// TwinCAT 3 PLC project PLC
// ProgramVersion: 3.1.4026.12
// CompilerDefines: VISU_USEPROPERTYINFO
// libraries:
//   Tc2_MC2, * (Beckhoff Automation GmbH)
//   Tc2_SPA, * (Beckhoff Automation GmbH)
//   Tc2_Standard, * (Beckhoff Automation GmbH)
//   Tc2_System, * (Beckhoff Automation GmbH)
//   Tc2_Utilities, * (Beckhoff Automation GmbH)
//   VisuSymbols, 4.5.0.0 (System)
// project tree:
//   / GlobalTextList.TcGTLO, PlcTask.TcTTO, Visualization Manager.TcVMO (not stored)
//   GVLs/ GVL.TcGVL
//   POUs/ FB_PositionMotors.TcPOU, FB_PyListener.TcPOU, MAIN.TcPOU
//   VISUs/ Visualization.TcVIS
// real-time tasks:
//   TASK PlcTask: cycle T#10ms, priority 20, ADS port 350
// motion (NC):
//   TASK NC-Task 1 SAF: cycle T#2ms, priority 4, ADS port 501
//   TASK NC-Task 1 SVB: cycle T#10ms, priority 8, ADS port 511
//   AXIS Az (id 1)
//     General: UnitName=°, UnitFlags=#x00000004
//     OtherSettings: AllowMotionCmdToSlave=true
//     encoder EncType=1
//       Inc: RefSoftSyncMask=#x0000ffff
//     drive DrvType=5
//       Analog: TorqueSetpointScale=10, ScaleFactorActTorque=0.1
//       TimeComp: TaskDelayCycles=1
//     controller CtrType=1
//       CtrPara: PriorControlFactor=1
//         Observer: BandWidth=20
//   AXIS Alt (id 2)
//     General: UnitName=°, UnitFlags=#x00000004
//     PositionAreaControl: Enable=false
//     TargetPosControl: Enable=false
//     encoder EncType=1
//       SoftEndMinControl: Enable=true
//       SoftEndMaxControl: Enable=true, Range=90
//       Inc: RefSoftSyncMask=#x0000ffff
//     drive DrvType=5
//       Analog: TorqueSetpointScale=10, ScaleFactorActTorque=0.1
//       TimeComp: TaskDelayCycles=1
//     controller CtrType=1
//       CtrPara: PriorControlFactor=1
//         PosDiffControl: Enable=false
//         Observer: BandWidth=20
// I/O:
//   DEVICE Device 1 (EtherCAT), AmsNetId 192.168.1.5.2.1
//     Term 1 (EK1100) [EK1100 EtherCAT Coupler (2A E-Bus)]
//       Term 2 (EL7041) [EL7041 1Ch. Stepper motor output stage (50V, 5A)] (disabled)
//       Term 3 (EL7041) [EL7041 1Ch. Stepper motor output stage (50V, 5A)] (disabled)
// variable links:
//   PLC/PLC Instance <-> NC-Task 1 SAF/Axes/Alt
//     PlcTask Inputs/GVL.Alt.NcToPlc <-> Outputs/ToPlc
//     PlcTask Outputs/GVL.Alt.PlcToNc <-> Inputs/FromPlc
//   PLC/PLC Instance <-> NC-Task 1 SAF/Axes/Az
//     PlcTask Inputs/GVL.Az.NcToPlc <-> Outputs/ToPlc
//     PlcTask Outputs/GVL.Az.PlcToNc <-> Inputs/FromPlc

CONFIGURATION PLC
    RESOURCE PLC ON TwinCAT3
        TASK PlcTask(INTERVAL := T#10ms, PRIORITY := 20);
        PROGRAM MAIN WITH PlcTask : MAIN;
    END_RESOURCE
END_CONFIGURATION

// ---- GVLs/GVL.TcGVL
{attribute 'qualified_only'}
VAR_GLOBAL
	Alt				: Axis_Ref := Alt;
	Az				: Axis_Ref := Az;
END_VAR

// ---- POUs/MAIN.TcPOU
PROGRAM MAIN
VAR
	// Sun position variables
	fbGetTime				: NT_GetTime;
	fbPyListener			: FB_PyListener;
	currTime				: TIMESTRUCT;
	timer					: TON;
	fbSPA     				: FB_SPA;
    fSunZenith 				: LREAL;
    fSunAzimuth 			: LREAL;
	fSunAltitude			: LREAL;
    tSunrise    			: TIME;
    tSunset     			: TIME;
    eErrorCode 				: E_SPA_ErrorCode;
    bExecute    			: BOOL := TRUE;
    bInit     				: BOOL := TRUE;
	go						: BOOL := FALSE;
	
	// Motion control variables
	fbPositionMotors		: FB_PositionMotors;
	fbResetMotors			: MC_Reset;
	bResetMotors			: BOOL := FALSE;
	Az						: Axis_Ref;
	Alt						: Axis_Ref;
	
END_VAR

timer(
	IN := TRUE, 
	PT := T#1S
	);

fbGetTime(
	NETID := '',
	Start := timer.Q,
	TMOUT := DEFAULT_ADS_TIMEOUT,
	BUSY =>,
	ERRID =>,
	TIMESTR => currTime
	);
	
fbPylistener(bExecute := TRUE);					// Grab lat, long, and other data... tell the rest of the
												// program when its done and its good to go

IF timer.Q THEN
 	fbSPA.stTime.iYear := currTime.wYear;
 	fbSPA.stTime.iMonth := currTime.wMonth;
 	fbSPA.stTime.iDay := currtime.wDay;
 	fbSPA.stTime.iHour := currTime.wHour;
 	fbSPA.stTime.iMinute := currTime.wMinute;
 	fbSPA.fTimezone; 							// Uses UTC offset
 	fbSPA.fLongitude; 							// Grabbed from Python script
 	fbSPA.fLatitude; 							// Grabbed from Python script
 	fbSPA.fElevation; 							// Meters, grabbed from Python script
 	fbSPA.fTemperature := 20; 					// Celsius... grab temp from either web, python, USB, or whatever
 	fbSPA.eFunction := eSPA_ZA_RTS;
END_IF

IF go = TRUE THEN 								// Tie all GO commands to execute after geo location 
												// is found, Q timers

IF timer.Q THEN
	
    fbSPA();
	
    fSunZenith := fbSPA.fZenith;
	fSunAltitude := 90 - fSunZenith; 			// Get altitude from zenith
    fSunAzimuth := fbSPA.fAzimuth;
    tSunrise := LREAL_TO_TIME(fbSPA.fSunrise * 60 * 60 * 1000);
    tSunset := LREAL_TO_TIME(fbSPA.fSunset * 60 * 60 * 1000);
	
	eErrorCode := fbSPA.iErrorCode;
	
	fbPositionMotors( 
		fSunAltitude := fSunAltitude,
		fSunAzimuth := fSunAzimuth 
		);
	
	IF bResetMotors = TRUE THEN
		fbResetMotors(Axis := GVL.Az, Execute := TRUE);
		fbResetMotors(Axis := GVL.Alt, Execute := TRUE);
		bResetMotors := FALSE;
	END_IF
	
END_IF

IF (timer.Q) THEN
	timer(IN := FALSE);
END_IF

END_IF

END_PROGRAM

// ---- POUs/FB_PyListener.TcPOU
FUNCTION_BLOCK FB_PyListener
VAR_INPUT
	bExecute			: BOOL := FALSE;
	Initialized 		: BOOL := FALSE;
	Init_State  		: UINT := 0;
END_VAR
VAR_OUTPUT
	bIsBusy				: BOOL;
    ERR             	: BOOL;
    ERRID           	: UDINT;
END_VAR
VAR
	Process         	: NT_StartProcess;
	RisingEdge			: R_TRIG;
	bError          	: BOOL;
    sTargetFilePath     : STRING(255);
    sTargetDirectory    : STRING(255);
    sCommand        	: STRING(255);
    iErrorId            : UDINT; 	
END_VAR

IF NOT Initialized THEN
  (* Initialization State Machine *)
  CASE Init_State OF
    0: (* First step in initialization *)
	
		// File Locations
		sTargetDirectory := 'C:\Users\AEverman\Desktop\Celestial_Positioning\Celestial_Positioning\Celestial_Positioning\PLC\SCRIPTS\';
 
		// Build Command String                 
		// Special command indicating command string input
		sCommand := CONCAT(sTargetDirectory, 'GPS_COORD_FIND.py');      // Execute Python data collection script
        Init_State := Init_State + 1;
	   
    1: (* Second step in initialization *)
		Process(
    	NETID := '',                    					// Local System
		//PATHSTR := 'C:\ProgramData\Anaconda3\python.exe ',   // Path to local cmd executable
		PATHSTR := 'python',
    	COMNDLINE := sCommand,          					// Comnmand to be executed
    	ERR => bError,                   					// Error Output
    	ERRID => iErrorId,                					// Error Id Output
		BUSY => bIsBusy,									// Process is already busy, used to not call multiple instances
		START := TRUE
		);
        Init_State := Init_State + 1;

    2: (* Last step in initialization *)
		Process(
			START := FALSE,
			BUSY => bIsBusy
		);
		bExecute := FALSE;
		RisingEdge.CLK := FALSE;
        Initialized := TRUE;
  END_CASE
END_IF

END_FUNCTION_BLOCK

// ---- POUs/FB_PositionMotors.TcPOU
FUNCTION_BLOCK FB_PositionMotors
VAR_INPUT
	fSunAltitude		: LREAL;
	fSunAzimuth			: LREAL;
END_VAR
VAR_OUTPUT
	Done_Alt			: BOOL;
	Busy_Alt			: BOOL;
	Active_Alt			: BOOL;
	Error_Alt			: BOOL;
	ErrorID_Alt			: UDINT;
	
	Done_Az				: BOOL;
	Busy_Az				: BOOL;
	Active_Az			: BOOL;
	Error_Az			: BOOL;
	ErrorID_Az			: UDINT;
END_VAR
VAR
	Step				: INT := 0;	

	
	fbPowerAlt			: MC_Power;
	fbPowerAz			: MC_Power;
	fbMoveAlt			: MC_MoveAbsolute;
	fbMoveAz			: MC_MoveAbsolute;
	fbHaltAz			: Mc_Halt;
	fbHaltAlt			: Mc_Halt;
END_VAR

CASE step OF

0:	
fbPowerAlt(
	Axis := GVL.Alt,
	Enable := TRUE,
	Enable_Positive := TRUE,
	Enable_Negative := TRUE,
	Override := 100,
	);
	
fbPowerAz(
	Axis := GVL.Az,
	Enable := TRUE,
	Enable_Positive := TRUE,
	Enable_Negative := TRUE,
	Override := 100,
	);
	
	step := 1;

1:
fbMoveAlt(
	Axis := GVL.Alt,
	Execute := TRUE,
	Position := fSunAltitude,
	Velocity := 5,
	Acceleration := 1,
	Deceleration := 1,
	Jerk := 1,
	Done => Done_Alt,
	Busy => Busy_Alt,
	Active => Active_Alt,
	Error => Error_Alt,
	ErrorID => ErrorID_Alt,
	);
	
step := 2;

2:
fbMoveAz(
	Axis := GVL.Az,
	Execute := TRUE,
	Position := fSunAzimuth,
	Velocity := 5,
	Acceleration := 1,
	Deceleration := 1,
	Jerk := 1,
	Done => Done_Az,
	Busy => Busy_Az,
	Active => Active_Az,
	Error => Error_Az,
	ErrorID => ErrorID_Az,
	);
	
	step := 10;
3:	
fbHaltAlt(
	Axis := GVL.Alt,
	Execute := TRUE,
	Deceleration := 1,
	Jerk := 1,
	Done => Done_Alt,
	Busy => Busy_Alt,
	Active => Active_Alt
	);
	
	step := 4;

4:
fbHaltAz(
	Axis := GVL.Az,
	Execute := TRUE,
	Deceleration := 1,
	Jerk := 1,
	Done => Done_Az,
	Busy => Busy_Az,
	Active => Active_Az,
	);
	
step := 1;

10:
fbMoveAz.Execute := FALSE;
fbMoveAlt.Execute := FALSE;
step := 1;

END_CASE

END_FUNCTION_BLOCK

// ---- GlobalTextList.TcGTLO
TEXTLIST GlobalTextList
  953 = '%3.5'
  159 = '%3.5f'
  465 = '%f 3.5'
  15 = '%f3.5'
  345 = '%s'
  276 = '%s3.5'
  249 = '%tHHmmssms'
  154 = '%t[HH/mm/ss/ms]'
  917 = '%t[HHmmssms]'
  999 = '%t[yyyy/MM/dd  HH/mm/ss/ms]'
  117 = '%t[yyyy/MM/dd/HH/mm/ss/ms]'
  6 = 'Alt Error'
  361 = 'Az Error'
  929 = 'Clear Motor Faults'
  911 = 'Current Time'
  641 = 'Label'
  586 = 'Latitude'
  280 = 'Longitude'
  682 = 'Motor Alt'
  4 = 'Motor Az'
  592 = 'Solar Telescope Controls'
  167 = 'Solar Tracking Telescope Controls'
  907 = 'Sun Alt'
  633 = 'Sun Az'
  395 = 'Telescope Controls'
END_TEXTLIST

// ---- VISUs/Visualization.TcVIS
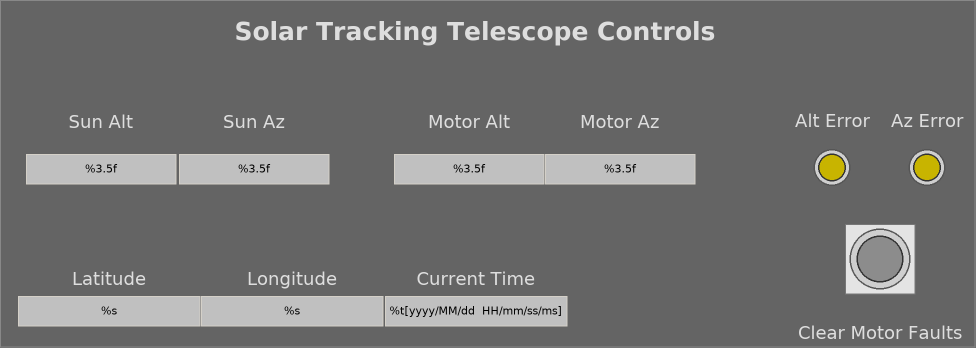
VISUALIZATION Visualization  // 976x348
    Label (217,5 516x52), "Solar Tracking Telescope Controls"
    Label (179,107 150x30), "Sun Az"
    Textfield (179,154 150x30), "%3.5f", text variable: MAIN.fSunAzimuth
    Label (26,107 150x30), "Sun Alt"
    Textfield (26,154 150x30), "%3.5f", text variable: MAIN.fSunAltitude
    Label (401,264 150x30), "Current Time"
    Textfield (385,296 182x30), "%t[yyyy/MM/dd HH/mm/ss/ms]", text variable: MAIN.currTime
    Textfield (545,154 150x30), "%3.5f", text variable: GVL.Az.NcToPlc.ActPos
    Label (545,107 150x30), "Motor Az"
    Textfield (394,154 150x30), "%3.5f", text variable: GVL.Alt.NcToPlc.ActPos
    Label (394,107 150x30), "Motor Alt"
    Label (34,264 150x30), "Latitude"
    Textfield (18,296 182x30), "%s", text variable: MAIN.fbSPA.fLatitude
    Label (217,264 150x30), "Longitude"
    Textfield (201,296 182x30), "%s", text variable: MAIN.fbSPA.fLongitude
    Group (785,106 190x83)
        Lamp1 (26,40 42x43), variable: MAIN.fbPositionMotors.Error_Alt, style: Lamp-Lamp1-Yellow
        Lamp1 (121,40 42x43), variable: MAIN.fbPositionMotors.Error_Az, style: Lamp-Lamp1-Yellow
        Label (0,0 95x30), "Alt Error"
        Label (95,0 95x30), "Az Error"
    PushSwitch (845,224 70x70), variable: MAIN.bResetMotors, behaviour: TOGGLE, style: Switch-PushSwitch-Gray
    Label (785,318 191x30), "Clear Motor Faults"
END_VISUALIZATION
